damping module: Internal overtemperature / HF-Dämpfungsmodul: Übertemperatur Innenraum'; 37040 'HF damping module: Undervoltage 24 V / HF-Dämpfungsmodul: Unterspannung 24 V'; 37041 'HF damping module: Undervoltage 24 V alarm / HF-Dämpfungsmodul: Unterspannung 24 V Warnung'; 37043 'HF damping module: Overvoltage 24 V / HF-Dämpfungsmodul: Überspannung 24 V'; 37044 'HF damping module: Overvoltage 24 V alarm / HF-Dämpfungsmodul: Überspannung 24 V Warnung'; 37045 'HF damping module: Undervoltage supply / HF-Dämpfungsmodul: Unterspannung Versorgung'; 37049 'Damping module: Internal fan faulty / Dämpfungsmodul: Innenraumlüfter defekt'; 37050 'HF damping module: Overvoltage 24 V fault / HF-Dämpfungsmodul: Überspannung 24 V Störung'; 37052 'HF damping module: EEPROM data error / HF-Dämpfungsmodul: EEPROM-Daten fehlerhaft'; 37056 'HF damping module: Heat sink overtemperature / HF-Dämpfungsmodul: Übertemperatur Kühlkörper'; 37310 'HF reactor module: Overtemperature / HF-Drosselmodul: Übertemperatur'; 37311 'HF reactor module: Overtemperature heat sink / HF-Drosselmodul: Übertemperatur Kühlkörper'; 37312 'HF reactor module: Overtemperature or fan failure / HF-Drosselmodul: Übertemperatur oder Lüfterausfall'; 37313 'HF reactor module: Overtemperature or fan failure / HF-Drosselmodul: Übertemperatur oder Lüfterausfall'; 37502 'HF damping module: Damping voltage too high / HF-Dämpfungsmodul: Dämpfungsspannung zu hoch'; 37800 'HF damping module: Group signal / HF-Dämpfungsmodul: Sammelmeldung'; 37801 'HF damping module: Sign of life missing / HF-Dämpfungsmodul: Lebenszeichen fehlt'; 37820 'HF damping module: Telegram error / HF-Dämpfungsmodul: Telegramm fehlerhaft'; 37835 'HF damping module: Cyclic data transmission error / HF-Dämpfungsmodul: Zyklische Datenübertragung gestört'; 37837 'HF damping module: Component faulted / HF-Dämpfungsmodul: Komponente gestört'; 37845 'HF damping module: Cyclic data transmission error / HF-Dämpfungsmodul: Zyklische Datenübertragung gestört'; 37850 'HF damping module: Internal software error / HF-Dämpfungsmodul: Softwarefehler intern'; 37851 'HF damping module (CU): Sign of life missing / HF-Dämpfungsmodul (CU): Lebenszeichen fehlt'; 37860 'HF damping module (CU): Telegram error / HF-Dämpfungsmodul (CU): Telegramm fehlerhaft'; 37885 'HF damping module (CU): Cyclic data transmission error / HF-Dämpfungsmodul (CU): Zyklische Datenübertragung gestört'; 37887 'HF damping module (CU): Component faulted / HF-Dämpfungsmodul (CU): Komponente gestört'; 37895 'HF damping module (CU): Alternating cyclic data transmission error HF-Dämpfungsmodul (CU): Alternierend zyklische Datenübertragung gestört'; 37896 'HF damping module (CU): Inconsistent component properties HF-Dämpfungsmodul (CU): Komponenteneigenschaften inkonsistent'; 37898 'HF damping module: POWER ON signal / HF-Dämpfungsmodul: POWER ON Meldung'; 37899 'HF damping module: Unknown fault / HF-Dämpfungsmodul: Unbekannte Störung'; 37903 'HF damping module: I2C bus error occurred / HF-Dämpfungsmodul: I2C-Bus Fehler aufgetreten'; 37999 'HF DM: Unknown alarm / HF-Dämpfungsmodul: Unbekannte Warnung'; 40799 'CX32: Configured transfer end time exceeded / CX32: Projektierter Transferendezeitpunkt überschritten'; 49200 'Excitation group signal fault / Erregung Sammelsignal Störung'; 49201 'Excitation group signal alarm / Erregung Sammelsignal Warnung'; 49920 'Protective breaker, main circuit tripped / Schutzschalter Hauptstromkreis ausgelöst'; 49921 'Protective breaker redundant main circuit tripped / Schutzschalter redundanter Hauptstromkreis ausgelöst'; 49922 'Protective breaker 24 V circuit has tripped / Schutzschalter 24-V-Stromkreis ausgelöst'; 49923 'Protective breaker terminal strip 24 V circuit has tripped / Schutzschalter Klemmenleiste 24-V-Stromkreis ausgelöst'; 49924 'Protective breaker power unit supply circuit tripped / Schutzschalter Leistungsteilversorgung Stromkreis ausgelöst'; 49926 'Protective breaker synchronizing voltage tripped / Schutzschalter Synchronisierspannung ausgelöst'; 49927 'Protective breaker auxiliary fan circuit has tripped / Schutzschalter Hilfslüfterstromkreis ausgelöst'; 49933 'Protective breaker excitation 230 V AC circuit tripped / Schutzschalter Erregung AC 230-V-Stromkreis ausgelöst'; 49934 'Protective breaker output cooling unit 230 V AC circuit tripped Schutzschalter Abgang Kühlanlage AC 230-V-Stromkreis ausgelöst'; 49935 'Protective breaker power unit door solenoids 24 V circuit has tripped Schutzschalter Leistungsteil Türmagnete 24-V-Stromkreis ausgelöst'; 49936 'Prot. breaker lighting supply/socket outlets 230V AC cct has tripped Schutzschalter Lichtnetz/Steckdosen AC 230-V-Stromkreis ausgelöst'; 49937 'UPS not ready / USV nicht bereit'; 49938 'UPS battery operation / USV Batteriebetrieb'; 49939 'UPS battery discharged / USV Batterie entladen'; 50001 'PROFINET configuration error / COMM BOARD: Alarm 1 / PROFINET Konfigurationsfehler / COMM BOARD: Warnung 1'; 50002 'COMM BOARD: Alarm 2 / COMM BOARD: Warnung 2'; 50003 'COMM BOARD: Alarm 3 / COMM BOARD: Warnung 3'; 50004 'COMM BOARD: Alarm 4 / COMM BOARD: Warnung 4'; 50005 'COMM BOARD: Alarm 5 / COMM BOARD: Warnung 5'; 50006 'COMM BOARD: Alarm 6 / COMM BOARD: Warnung 6'; 50007 'COMM BOARD: Alarm 7 / COMM BOARD: Warnung 7'; 50008 'COMM BOARD: Alarm 8 / COMM BOARD: Warnung 8'; 50009 'COMM BOARD: Alarm 9 / COMM BOARD: Warnung 9'; 50010 'COMM BOARD: Alarm 10 / COMM BOARD: Warnung 10'; 50011 'COMM BOARD: Alarm 11 / COMM BOARD: Warnung 11'; 50012 'COMM BOARD: Alarm 12 / COMM BOARD: Warnung 12'; 50013 'COMM BOARD: Alarm 13 / COMM BOARD: Warnung 13'; 50014 'COMM BOARD: Alarm 14 / COMM BOARD: Warnung 14'; 50015 'COMM BOARD: Alarm 15 / COMM BOARD: Warnung 15'; 50016 'COMM BOARD: Alarm 16 / COMM BOARD: Warnung 16'; 50017 'COMM BOARD: Alarm 17 / COMM BOARD: Warnung 17'; 50018 'COMM BOARD: Alarm 18 / COMM BOARD: Warnung 18'; 50019 'COMM BOARD: Alarm 19 / COMM BOARD: Warnung 19'; 50020 'PROFINET: Second controller missing / COMM BOARD: Alarm 20 PROFINET: Zweiter Controller fehlt / COMM BOARD: Warnung 20'; 50201 'COMM BOARD: Fault 1 / COMM BOARD: Störung 1'; 50202 'COMM BOARD: Fault 2 / COMM BOARD: Störung 2'; 50203 'COMM BOARD: Fault 3 / COMM BOARD: Störung 3'; 50204 'COMM BOARD: Fault 4 / COMM BOARD: Störung 4'; 50205 'COMM BOARD: Fault 5 / COMM BOARD: Störung 5'; 50206 'COMM BOARD: Fault 6 / COMM BOARD: Störung 6'; 50207 'COMM BOARD: Fault 7 / COMM BOARD: Störung 7'; 50208 'COMM BOARD: Fault 8 / COMM BOARD: Störung 8'; 50209 'COMM BOARD: Fault 9 / COMM BOARD: Störung 9'; 50210 'COMM BOARD: Fault 10 / COMM BOARD: Störung 10'; 50211 'COMM BOARD: Fault 11 / COMM BOARD: Störung 11'; 50212 'COMM BOARD: Fault 12 / COMM BOARD: Störung 12'; 50213 'COMM BOARD: Fault 13 / COMM BOARD: Störung 13'; 50214 'COMM BOARD: Fault 14 / COMM BOARD: Störung 14'; 50215 'COMM BOARD: Fault 15 / COMM BOARD: Störung 15'; 50216 'No texts available / Kein Text verfügbar'

Template "Template_1" 480x272
   Button "Exit" at 388,227 size 63x44; TextOff 'Exit'; PictureOff "ExitRuntime_KTP400_Basic_PN_TR"; PictureOn "ExitRuntime_KTP400_Basic_PN_TR"
      on Release: StopRuntime(0)
   Button "Template_Button" at 268,227 size 63x44; TextOff 'Text'
   Button "Alarms" at 148,227 size 63x44; TextOff 'Alarms'; PictureOff "AlarmDisplay_KTP400_Basic_PN_TR"; PictureOn "AlarmDisplay_KTP400_Basic_PN_TR"
      on Release: function_ef3f5d25("Alarm window_Unacknowledged", -1)
   Button "Start screen" at 28,227 size 63x44; TextOff 'Start screen'; PictureOff "NavigateHome_KTP400_Basic_PN_TR"; PictureOn "NavigateHome_KTP400_Basic_PN_TR"
      on Release: ActivateScreen("Root screen", 0)
   SymbolicIOField "Symbolic_IO_Field_Screen" at 82,8 size 311x29; TextOff '0'; TextOn '1'; TextList "TextList_ScreenNames"
      ProcessValue <- "Tag_ScreenNumber"
      on Change: ActivateScreenByNumber("Tag_ScreenNumber", 0)
   DateTimeField "HmiScreenItemData" at 395,22 size 85x22
   DateTimeField "HmiScreenItemData_1" at 395,0 size 85x22
   GraphicView "Logo" at 0,0 size 80x45; Picture "Logo of HMI_1"

screen "Root screen" 480x272
   on GenerateScreen: SetTag("Tag_ScreenNumber", 1)
   TextField "HmiScreenItemData" at 6,68 size 469x22; Text 'Upravljanje sinhronim reluktantnim motorom'
   Button "Screen0" at 1,170 size 157x30; TextOff 'Upravljanje brzinom'; TextOn 'Screen0'
      on Release: ActivateScreen("Screen0", 0)
   Button "Screen1" at 162,170 size 157x30; TextOff 'Prikaz momenta'; TextOn 'Screen1'
      on Release: ActivateScreen("Screen1", 0)
   Button "Screen2" at 322,170 size 157x30; TextOff 'Prikaz struje'; TextOn 'Screen2'
      on Release: ActivateScreen("Screen2", 0)
   TextField "Text field_1" at 127,112 size 225x23; Text 'Student: Hažiabdić Merima'

screen "Screen0" 480x272
   on GenerateScreen: SetTag("Tag_ScreenNumber", 2)
   Button "Back" at 4,3 size 82x30; TextOff 'Nazad'; TextOn 'Back'
      on Release: ActivateScreen("Root screen", 0)
   TextField "Text field_1" at 7,39 size 65x25; Text 'Brzina:'
   IOField "I/O field_1" at 86,37 size 96x32; FormatPattern 9999
      ProcessValue <- "zadanaPID"
   TextField "Text field_2" at 190,39 size 44x25; Text 'Rpm'
   TrendView "Trend view_1" at 0,76 size 480x196
   Switch "Switch_1" at 256,20 size 96x32; CaptionText 'Switch'; TextOff 'START'; TextOn 'STOP'; PictureOff "START"
      on SwitchOn: SetBit("ON_OFF1")
      on SwitchOff: ResetBit("ON_OFF1")
      Appearance <- "ON_OFF1"
      ProcessValue <- "ON_OFF1"
   Switch "Switch_2" at 373,20 size 96x32; CaptionText 'Switch'; TextOff 'DESNO'; TextOn 'LIJEVO'; PictureOff "Graphic_1"
      ProcessValue <- "Dir_rev"
      on SwitchOn: SetBit("Dir_rev")
      on SwitchOff: ResetBit("Dir_rev")

screen "Screen1" 480x272
   on GenerateScreen: SetTag("Tag_ScreenNumber", 3)
   TextField "HmiScreenItemData" at 55,7 size 373x22; Text 'Prikaz momenta'
   Button "Back" at 4,3 size 82x30; TextOff 'Nazad'; TextOn 'Back'
      on Release: ActivateScreen("Root screen", 0)
   TrendView "Trend view_1" at 0,39 size 480x233

screen "Screen2" 480x272
   on GenerateScreen: SetTag("Tag_ScreenNumber", 4)
   TextField "HmiScreenItemData" at 56,7 size 373x22; Text 'Prikaz struje'
   Button "Back" at 4,3 size 82x30; TextOff 'Nazad'; TextOn 'Back'
      on Release: ActivateScreen("Root screen", 0)
   TrendView "Trend view_1" at 0,40 size 480x232

screen "Screen_1" 480x272
   Button "Button_1" at 12,8 size 96x32; TextOff 'on'
      on Click: InvertBit("ON_OFF1")
   Button "Button_2" at 143,10 size 96x32; TextOff 'off2'
      on Click: InvertBit("OFF2")
   Button "Button_3" at 277,17 size 96x32; TextOff 'off3'
      on Click: InvertBit("OFF3")
   Button "Button_4" at 384,13 size 96x32; TextOff 'ack'
      on Click: InvertBit("Ack")
   Button "Button_5" at 25,69 size 96x32; TextOff 'rev'
      on Click: InvertBit("Dir_rev")
   Button "Button_6" at 148,71 size 96x32; TextOff '0'
      on Click: InvertBit("Reset_SP")
   Button "Button_7" at 269,74 size 96x32; TextOff 'n+'
      on Click: InvertBit("Inc_SP")
   Button "Button_8" at 379,77 size 96x32; TextOff 'n-'
      on Click: InvertBit("Dec_SP")
   Button "Button_9" at 78,158 size 96x32; TextOff 'Nazad'
      on Release: ActivateScreen("Root screen", 0)
*)